{attribute 'enable_dynamic_creation'}
FUNCTION_BLOCK TestNode IMPLEMENTS ITF_Node
VAR
	_next : ITF_Node;
    _prev : ITF_Node;
    _pos  : UINT;
END_VAR

METHOD GetLastNode : ITF_Node
GetLastNode := _prev;
END_METHOD

METHOD GetMyPointer : PVOID
GetMyPointer := ADR(THIS^);
END_METHOD

METHOD GetNextNode : ITF_Node
GetNextNode := _next;
END_METHOD

METHOD GetPositionInList : UINT
GetPositionInList := _pos;
END_METHOD

METHOD SetLastNode : BOOL
VAR_INPUT
	Node	: ITF_Node;
END_VAR
_prev := Node; 

SetLastNode := TRUE;
END_METHOD

METHOD SetNextNode : BOOL
VAR_INPUT
	Node	: ITF_Node;
END_VAR
_next := Node; 

SetNextNode := TRUE;
END_METHOD

METHOD SetPositionInList : BOOL
VAR_INPUT
	Index	: UINT;
END_VAR
_pos := Index; 

SetPositionInList := TRUE;
END_METHOD

END_FUNCTION_BLOCK

(* stored: Version 1.1.0.1
   POU TestNode: Id {0bcb7e1e-127a-43ae-bea2-b98dab94b334}, SpecialFunc None
   Method GetLastNode: Id {253d8c54-70d8-4367-86f8-d532631c4b16}
   Method GetMyPointer: Id {19e406ff-acf2-4b69-bccb-f8bd4ad3075d}
   Method GetNextNode: Id {5d013b56-826c-404c-8b9a-ffb51d84435b}
   Method GetPositionInList: Id {7676de77-38f7-4e44-a0a5-02e4079f2f99}
   Method SetLastNode: Id {b28a873d-7080-434a-b3b7-113729e08fe4}
   Method SetNextNode: Id {6f500d5a-1898-4f98-a0f9-160b1b0fe1de}
   Method SetPositionInList: Id {887ab231-72a1-41d8-901a-3cdbe41f8e5a} *)
